// TIA Portal V19 export
DATA_BLOCK "SET PARAMETER DB"   // DB44
{ S7_Optimized_Access := 'TRUE' }
// stored: MemoryReserve 100
   VAR RETAIN
      "MANUAL VFD SET PARAMETER" : Struct
         "MFG VESSEL STIRROR RUN" : Real;
         "PREMIXING  VESSEL STIRROR RUN" : Real;
         "SUGAR VESSEL STIRROR RUN" : Real;
      END_STRUCT;
   END_VAR
   VAR
      "AUTO VFD SET PARAMETER" : Struct
         "MFG VESSEL STIRROR RUN" : Real;
         "PREMIXING  VESSEL STIRROR RUN" : Real;
         "SUGAR VESSEL STIRROR RUN" : Real;
      END_STRUCT;
   END_VAR
BEGIN
END_DATA_BLOCK
